// TwinCAT 3 PLC project RunnerLib
// Title: Runner Library
// Company: Beckhoff UK
// Author: Chris Knight
// ProjectVersion: 2.0.0.0
// ProgramVersion: 3.1.4026.14
// libraries:
//   Base Library, * (Beckhoff UK)
//   Tc2_Standard, * (Beckhoff Automation GmbH)
//   Tc2_System, * (Beckhoff Automation GmbH)
//   Tc3_Module, * (Beckhoff Automation GmbH)
// project tree:
//   Cyclic Runner/ I_Object.TcIO, I_HostObjects.TcIO, ObjectRunner.TcPOU

// ---- Cyclic Runner/I_Object.TcIO
INTERFACE I_Object

METHOD RegisterWithParent
VAR_INPUT
	Runner : I_HostObjects;
END_VAR
END_METHOD

END_INTERFACE

// ---- Cyclic Runner/I_HostObjects.TcIO
INTERFACE I_HostObjects

METHOD DeregisterAllModules : HRESULT
VAR_INPUT
END_VAR
END_METHOD

METHOD RegisterAbortable : HRESULT
VAR_INPUT
	Abortable : I_Abortable;
END_VAR
END_METHOD

METHOD RegisterCyclic : HRESULT
VAR_INPUT
	Cyclic : I_Cyclic;
END_VAR
END_METHOD

METHOD RegisterInitialise : HRESULT
VAR_INPUT
	Initialise : I_Initialisable;
END_VAR
END_METHOD

METHOD RegisterResettable : HRESULT
VAR_INPUT
	Resetable : I_Resettable;
END_VAR
END_METHOD

END_INTERFACE

// ---- Cyclic Runner/ObjectRunner.TcPOU
FUNCTION_BLOCK ObjectRunner IMPLEMENTS I_Cyclic, I_HostObjects
VAR_INPUT
END_VAR
VAR_OUTPUT
END_VAR
VAR
	CyclicModules : ARRAY[0..MaxRegisteredModules] OF I_Cyclic;
	InitialiseModules : ARRAY[0..MaxRegisteredModules] OF I_Initialisable;
	ResetableModules : ARRAY[0..MaxRegisteredModules] OF I_Resettable;
	AbortableModules : ARRAY[0..MaxRegisteredModules] OF I_Abortable;
	CyclicModuleCount : INT := 0;
	InitModuleCount : INT := 0;
	ResetModuleCount : INT := 0;
	i: INT;
	InitialisationCount : INT := 0;
	Registered: BOOL;
	Initialised : BOOL := FALSE;
	AbortModuleCount: INT;
END_VAR
VAR CONSTANT
	MaxRegisteredModules : INT := 99;
END_VAR

METHOD AreAllModuleInitialised : BOOL
VAR_INPUT
END_VAR
AreAllModuleInitialised := Initialised;
END_METHOD

METHOD PUBLIC  Cycle : HRESULT
VAR_INPUT
END_VAR
FOR i := 0 TO MaxRegisteredModules DO
	IF CyclicModules[i] <> 0 THEN
		CyclicModules[i].Cycle();
	END_IF
END_FOR
END_METHOD

METHOD DeregisterAllModules : HRESULT
VAR_INPUT
END_VAR
FOR i := 0 TO MaxRegisteredModules DO
	CyclicModules[i] := 0;
	InitialiseModules[i] := 0;
	ResetableModules[i] := 0;
END_FOR
CyclicModuleCount := 0;
InitModuleCount := 0;
ResetModuleCount := 0;
DeregisterAllModules := S_OK;
END_METHOD

METHOD GetCyclicModuleCount : INT
VAR_INPUT
END_VAR
GetCyclicModuleCount := CyclicModuleCount;
END_METHOD

METHOD GetInitModuleCount : INT
VAR_INPUT
END_VAR
GetInitModuleCount := InitModuleCount;
END_METHOD

METHOD GetResetableModuleCount : INT
VAR_INPUT
END_VAR
GetResetableModuleCount := ResetModuleCount;
END_METHOD

METHOD Initialise : HRESULT
VAR_INPUT
END_VAR
IF InitialisationCount = 0 THEN
	Initialised := TRUE;
	Initialise := S_FALSE;
ELSE
	IF InitialisationCount < MaxRegisteredModules THEN
		IF InitialiseModules[InitialisationCount] <> 0 THEN
			IF InitialiseModules[InitialisationCount].Initialise() = 2 THEN
				InitialisationCount := InitialisationCount + 1;
			END_IF
		ELSE
			InitialisationCount := InitialisationCount + 1;
		END_IF
	ELSE
		Initialise := S_OK;
		InitialisationCount := 0;
		Initialised := TRUE;
	END_IF
END_IF
END_METHOD

METHOD RegisterAbortable : HRESULT
VAR_INPUT
	Abortable : I_Abortable;
END_VAR
IF Abortable <> 0 AND_THEN AbortModuleCount < (MaxRegisteredModules + 1) THEN
	Registered := FALSE;
	FOR i := 0 TO MaxRegisteredModules DO
		IF AbortableModules[i] = Abortable THEN
			Registered := TRUE;
		END_IF
	END_FOR
	IF NOT Registered THEN	
		FOR i := 0 TO MaxRegisteredModules DO
			IF AbortableModules[i] = 0 THEN
				AbortableModules[i] := Abortable;
				AbortModuleCount := AbortModuleCount + 1;
				EXIT;
			END_IF
		END_FOR
		RegisterAbortable := 1;
	ELSE
		RegisterAbortable := -1;
	END_IF	
ELSE
	RegisterAbortable := -2;
END_IF
END_METHOD

METHOD RegisterCyclic : HRESULT
VAR_INPUT
	Cyclic : I_Cyclic;
END_VAR
IF Cyclic <> 0 AND_THEN CyclicModuleCount < (MaxRegisteredModules + 1) THEN
	Registered := FALSE;
	FOR i := 0 TO MaxRegisteredModules DO
		IF CyclicModules[i] = Cyclic THEN
			Registered := TRUE;
		END_IF
	END_FOR
	IF NOT Registered THEN	
		FOR i := 0 TO MaxRegisteredModules DO
			IF CyclicModules[i] = 0 THEN
				CyclicModules[i] := Cyclic;
				CyclicModuleCount := CyclicModuleCount + 1;
				EXIT;
			END_IF
		END_FOR
		RegisterCyclic := 1;
	ELSE
		RegisterCyclic := -1;
	END_IF	
ELSE
	RegisterCyclic := -2;
END_IF
END_METHOD

METHOD RegisterInitialise : hresult
VAR_INPUT
	Initialise : I_Initialisable;
END_VAR
IF Initialise <> 0 AND_THEN CyclicModuleCount < (MaxRegisteredModules + 1) THEN
	Registered := FALSE;
	FOR i := 0 TO MaxRegisteredModules DO
		IF InitialiseModules[i] = Initialise THEN
			Registered := TRUE;
		END_IF
	END_FOR
	IF NOT Registered THEN	
		FOR i := 0 TO MaxRegisteredModules DO
			IF InitialiseModules[i] = 0 THEN
				InitialiseModules[i] := Initialise;
				InitModuleCount := InitModuleCount + 1;
			END_IF
			EXIT;
		END_FOR
		RegisterInitialise := 1;
	ELSE
		RegisterInitialise := -1;
	END_IF	
ELSE
	RegisterInitialise := -2;
END_IF
END_METHOD

METHOD RegisterModule : HRESULT
VAR_INPUT
	Registerable : I_Object;
END_VAR
IF Registerable <> 0 THEN
	Registerable.RegisterWithParent(THIS^);
	RegisterModule := 1;
ELSE
	RegisterModule := -1;
END_IF
END_METHOD

METHOD RegisterResettable : HRESULT
VAR_INPUT
	Resetable : I_Resettable;
END_VAR
IF Resetable <> 0 AND_THEN ResetModuleCount < (MaxRegisteredModules + 1) THEN
	Registered := FALSE;
	FOR i := 0 TO MaxRegisteredModules DO
		IF ResetableModules[i] = Resetable THEN
			Registered := TRUE;
		END_IF
	END_FOR
	IF NOT Registered THEN	
		FOR i := 0 TO MaxRegisteredModules DO
			IF ResetableModules[i] = 0 THEN
				ResetableModules[i] := Resetable;
				ResetModuleCount := ResetModuleCount + 1;
				EXIT;
			END_IF
		END_FOR
		RegisterResettable := 1;
	ELSE
		RegisterResettable := -1;
	END_IF	
ELSE
	RegisterResettable := -2;
END_IF
END_METHOD

END_FUNCTION_BLOCK
